// TIA Portal V19 export
FUNCTION_BLOCK "LEXCHANGETRAY_PressureGaugeRs485"   // FB557, LAD
TITLE = PressureGaugeRs485
AUTHOR : MR
// PressureGaugeRs485
// stored: Access Published, IsIECCheckEnabled true, MemoryReserve 100, SetENOAutomatically false
   VAR_IN_OUT
      getValue_sp3_1 : Array[0..2] of DInt;   // Function/variable to retrieve value from SP3_1
      getValue_sp4_1 : Array[0..2] of DInt;   // Function/variable to retrieve value from SP4_1
      controlNode : "typePressureGuageRs485ControlNode";   // Node for controlling system operations
      hmiInterface : "typePressureGuageRs485Interface";   // Interface for Human-Machine Interaction
      step_rs485 { ExternalAccessible := 'False'; ExternalVisible := 'False'; ExternalWritable := 'False'} : Int;   // Step configuration or status for RS485 communication
      writeMode { ExternalAccessible := 'False'; ExternalVisible := 'False'; ExternalWritable := 'False'} : Bool;   // Mode configuration for write operations
   END_VAR
   VAR
      statUp { ExternalAccessible := 'False'; ExternalVisible := 'False'; ExternalWritable := 'False'} : Bool;   // System uptime status flag
      statCommLoad { ExternalAccessible := 'False'; ExternalVisible := 'False'; ExternalWritable := 'False'} : Struct   // Communication load statistics structure
         done : Bool;
         error : Bool;
      END_STRUCT;
      statStatusSp1_1 { ExternalAccessible := 'False'; ExternalVisible := 'False'; ExternalWritable := 'False'} : Struct   // Status structure for SP1_1
         getDone : Bool;
         getBusy : Bool;
         getError : Bool;
         putDone : Bool;
         putBusy : Bool;
         putError : Bool;
      END_STRUCT;
      statStatusSp2_1 { ExternalAccessible := 'False'; ExternalVisible := 'False'; ExternalWritable := 'False'} : Struct   // Status structure for SP2_1
         getDone : Bool;
         getBusy : Bool;
         getError : Bool;
         putDone : Bool;
         putBusy : Bool;
         putError : Bool;
      END_STRUCT;
      statStatusSp3_1 { ExternalAccessible := 'False'; ExternalVisible := 'False'; ExternalWritable := 'False'} : Struct   // Status structure for SP3_1
         getDone : Bool;
         getBusy : Bool;
         getError : Bool;
         putDone : Bool;
         putBusy : Bool;
         putError : Bool;
      END_STRUCT;
      statStatusSp4_1 { ExternalAccessible := 'False'; ExternalVisible := 'False'; ExternalWritable := 'False'} : Struct   // Status structure for SP4_1
         getDone : Bool;
         getBusy : Bool;
         getError : Bool;
         putDone : Bool;
         putBusy : Bool;
         putError : Bool;
      END_STRUCT;
      instModbusCommLoad { ExternalAccessible := 'False'; ExternalVisible := 'False'; ExternalWritable := 'False'; S7_SetPoint := 'True'} : Modbus_Comm_Load;   // Modbus communication load instance
      instModbusMaster { ExternalAccessible := 'False'; ExternalVisible := 'False'; ExternalWritable := 'False'; S7_SetPoint := 'True'} : Modbus_Master;   // Modbus master instance configuration
   END_VAR
   VAR CONSTANT
      STEP1 : Int := 1;
      STEP2 : Int := 2;
      STEP3 : Int := 3;
      STEP4 : Int := 4;
      STEP5 : Int := 5;
      STEP6 : Int := 6;
      STEP7 : Int := 7;
      STEP8 : Int := 8;
      STEP9 : Int := 9;
      STEP10 : Int := 10;
      STEP11 : Int := 11;
      STEP12 : Int := 12;
      STEP13 : Int := 13;
      STEP14 : Int := 14;
      STEP15 : Int := 15;
      STEP16 : Int := 16;
      STEP17 : Int := 17;
      STEP18 : Int := 18;
      BAUD : UDInt := 19200;
      PARITY : UInt := 0;
      MB_ADDR_1 : UInt := 1;
      MB_ADDR_2 : UInt := 2;
      MB_ADDR_3 : UInt := 3;
      MB_ADDR_4 : UInt := 4;
      MODE_READ : USInt := 0;
      MODE_WRITE : USInt := 1;
      DATA_ADDR : UDInt := 40421;
      DATA_LEN_READ : UInt := 2;
   END_VAR
BEGIN

REGION Network 1 (SCL): 假的程序后续需要修改
   #hmiInterface.monitoring.simulation := #controlNode.commands.simulation;
   #hmiInterface.monitoring.enable := #controlNode.commands.quality;
END_REGION

REGION Network 2: step 3 SP3_1 Get pressure value
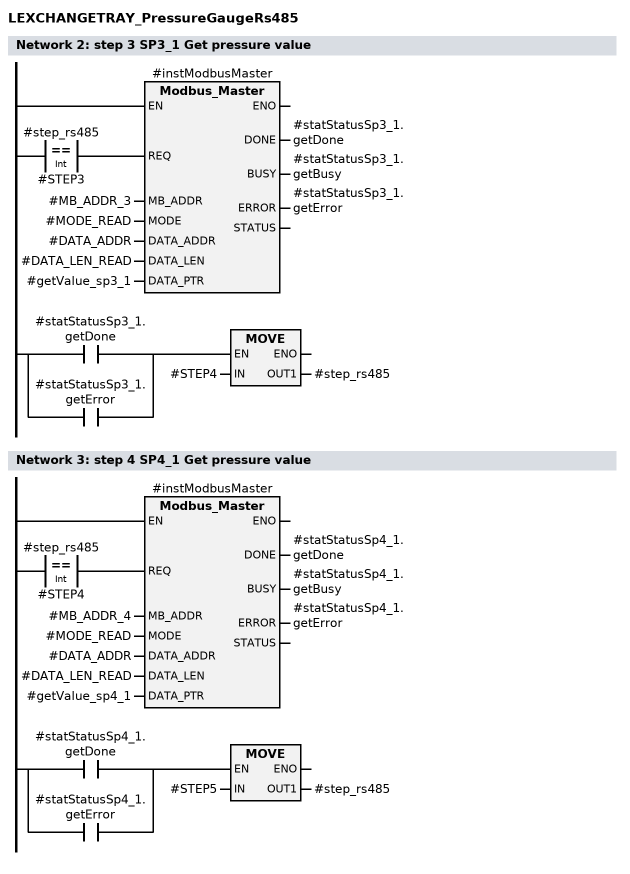
   RUNG wire#powerrail
      #instModbusMaster.Modbus_Master(REQ := wire#w1, MB_ADDR := #MB_ADDR_3, MODE := #MODE_READ, DATA_ADDR := #DATA_ADDR, DATA_LEN := #DATA_LEN_READ, DATA_PTR := #getValue_sp3_1, DONE => #statStatusSp3_1.getDone, BUSY => #statStatusSp3_1.getBusy, ERROR => #statStatusSp3_1.getError, STATUS =>)
   END_RUNG
   RUNG wire#powerrail
      { S7_Templates := "SrcType := Int" } EQ_Contact(in1 := #step_rs485, in2 := #STEP3)
   END_RUNG wire#w1
   RUNG wire#powerrail
      Contact( #statStatusSp3_1.getDone )
      wire#w2
      Move(in := #STEP4, out1 => #step_rs485)
   END_RUNG
   RUNG wire#powerrail
      Contact( #statStatusSp3_1.getError )
   END_RUNG wire#w2
   // the same network as SCL:
   #instModbusMaster(REQ := #step_rs485 = #STEP3,   // Modbus_Master
                     MB_ADDR := #MB_ADDR_3,
                     MODE := #MODE_READ,
                     DATA_ADDR := #DATA_ADDR,
                     DATA_LEN := #DATA_LEN_READ,
                     DATA_PTR := #getValue_sp3_1,
                     DONE => #statStatusSp3_1.getDone,
                     BUSY => #statStatusSp3_1.getBusy,
                     ERROR => #statStatusSp3_1.getError);
   IF #statStatusSp3_1.getDone OR #statStatusSp3_1.getError THEN #step_rs485 := #STEP4; END_IF;
END_REGION

REGION Network 3: step 4 SP4_1 Get pressure value
   RUNG wire#powerrail
      #instModbusMaster.Modbus_Master(REQ := wire#w1, MB_ADDR := #MB_ADDR_4, MODE := #MODE_READ, DATA_ADDR := #DATA_ADDR, DATA_LEN := #DATA_LEN_READ, DATA_PTR := #getValue_sp4_1, DONE => #statStatusSp4_1.getDone, BUSY => #statStatusSp4_1.getBusy, ERROR => #statStatusSp4_1.getError, STATUS =>)
   END_RUNG
   RUNG wire#powerrail
      { S7_Templates := "SrcType := Int" } EQ_Contact(in1 := #step_rs485, in2 := #STEP4)
   END_RUNG wire#w1
   RUNG wire#powerrail
      Contact( #statStatusSp4_1.getDone )
      wire#w2
      Move(in := #STEP5, out1 => #step_rs485)
   END_RUNG
   RUNG wire#powerrail
      Contact( #statStatusSp4_1.getError )
   END_RUNG wire#w2
   // the same network as SCL:
   #instModbusMaster(REQ := #step_rs485 = #STEP4,   // Modbus_Master
                     MB_ADDR := #MB_ADDR_4,
                     MODE := #MODE_READ,
                     DATA_ADDR := #DATA_ADDR,
                     DATA_LEN := #DATA_LEN_READ,
                     DATA_PTR := #getValue_sp4_1,
                     DONE => #statStatusSp4_1.getDone,
                     BUSY => #statStatusSp4_1.getBusy,
                     ERROR => #statStatusSp4_1.getError);
   IF #statStatusSp4_1.getDone OR #statStatusSp4_1.getError THEN #step_rs485 := #STEP5; END_IF;
END_REGION
END_FUNCTION_BLOCK
